// TIA Portal V17 export
// export: Created 2021-09-08T12:46:16.1780561Z, ExportSetting WithDefaults, DisplayName Totally Integrated Automation Portal, DisplayVersion V17, DisplayName TIA Portal Openness, DisplayVersion V17, DisplayName TIA Portal Version Control Interface, DisplayVersion V17, DisplayName STEP 7 Professional, DisplayVersion V17, DisplayName STEP 7 Safety, DisplayVersion V17, DisplayName WinCC Advanced, DisplayVersion V17
FUNCTION "SimplyMultiply" : Void   // FC11, LAD
{ S7_Optimized_Access := 'TRUE' }
VERSION : 1.1
// stored: AutoNumber true, IsIECCheckEnabled false, SetENOAutomatically false, StructureModified 2022-04-28T20:05:52, UDAEnableTagReadback false
   VAR_INPUT
      IN1 : Real;
      IN2 : Real;
   END_VAR
   VAR_OUTPUT
      Result : Real;
   END_VAR
BEGIN

REGION Network 1
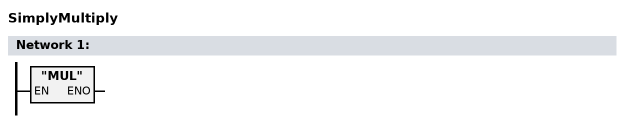
   RUNG wire#powerrail
      "MUL"()
   END_RUNG
   // the same network as SCL:
   "MUL"();
END_REGION
END_FUNCTION
